SUBAPPLICATION Schneidwerk (* Subapplication Type *)
  (* Standard: 61499-2 *)
  (* Version 1.0, 2023-01-29, Franz *)
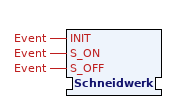
  EVENT_INPUT
    INIT;
    S_ON;
    S_OFF;
  END_EVENT
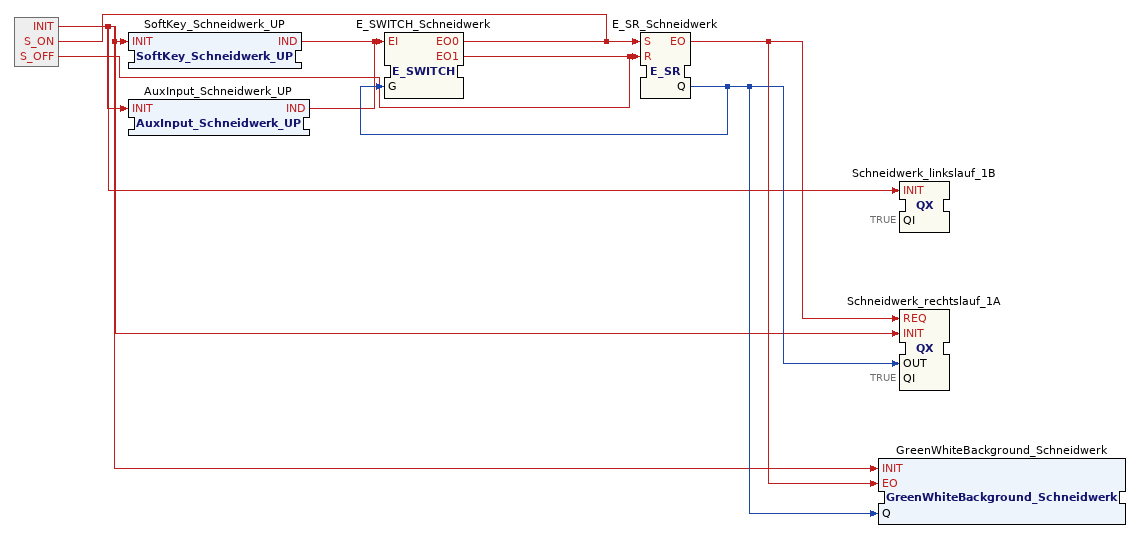
  FBS
    Schneidwerk_rechtslauf_1A : QX(QI := TRUE);
    E_SWITCH_Schneidwerk : E_SWITCH;
    E_SR_Schneidwerk : E_SR;
    Schneidwerk_linkslauf_1B : QX(QI := TRUE);
  END_FBS
  SUBAPPS
    SoftKey_Schneidwerk_UP : SoftKey_Schneidwerk_UP;
    GreenWhiteBackground_Schneidwerk : GreenWhiteBackground_Schneidwerk;
    AuxInput_Schneidwerk_UP : AuxInput_Schneidwerk_UP;
  END_SUBAPPS
  EVENT_CONNECTIONS
    E_SR_Schneidwerk.EO TO Schneidwerk_rechtslauf_1A.REQ;
    E_SWITCH_Schneidwerk.EO0 TO E_SR_Schneidwerk.S;
    E_SWITCH_Schneidwerk.EO1 TO E_SR_Schneidwerk.R;
    S_ON TO E_SR_Schneidwerk.S;
    S_OFF TO E_SR_Schneidwerk.R;
    INIT TO Schneidwerk_linkslauf_1B.INIT;
    INIT TO Schneidwerk_rechtslauf_1A.INIT;
    INIT TO SoftKey_Schneidwerk_UP.INIT;
    SoftKey_Schneidwerk_UP.IND TO E_SWITCH_Schneidwerk.EI;
    INIT TO GreenWhiteBackground_Schneidwerk.INIT;
    E_SR_Schneidwerk.EO TO GreenWhiteBackground_Schneidwerk.EO;
    AuxInput_Schneidwerk_UP.IND TO E_SWITCH_Schneidwerk.EI;
    INIT TO AuxInput_Schneidwerk_UP.INIT;
  END_CONNECTIONS
  DATA_CONNECTIONS
    E_SR_Schneidwerk.Q TO Schneidwerk_rechtslauf_1A.OUT;
    E_SR_Schneidwerk.Q TO E_SWITCH_Schneidwerk.G;
    E_SR_Schneidwerk.Q TO GreenWhiteBackground_Schneidwerk.Q;
  END_CONNECTIONS
END_SUBAPPLICATION
